// TIA Portal V17 export
// export: Created 2024-08-29T18:23:43.8090158Z, ExportSetting WithDefaults, DisplayName Totally Integrated Automation Portal, DisplayVersion V17 Update 7, DisplayName TIA Portal Openness, DisplayVersion V17 Update 7, DisplayName TIA Portal Version Control Interface, DisplayVersion V17, DisplayName SINAMICS Startdrive Advanced, DisplayVersion V17 SP2, DisplayName SINAMICS Startdrive G110M, G120, G120C, G120D, G120P, G115D, DisplayVersion V17 SP2, DisplayName SINAMICS Startdrive G130, G150, S120, S150, SINAMICS MV, S210, DisplayVersion V17 SP2, DisplayName STEP 7 Professional, DisplayVersion V17 Update 7, DisplayName STEP 7 Safety, DisplayVersion V17 Update 6, DisplayName WinCC Advanced / Unified PC, DisplayVersion V17 Update 7
DATA_BLOCK "analog"   // DB3
{ S7_Optimized_Access := 'TRUE' }
VERSION : 0.1
// stored: AutoNumber false, DBAccessibleFromOPCUA true, DBAccessibleFromWebserver true, IsOnlyStoredInLoadMemory false, IsRetainMemResEnabled false, IsWriteProtectedInAS false, MemoryReserve 100
   VAR RETAIN
      value1 : Array[0..32] of Real;   // Setpoint del valor analógico 1 [modelo]
      low1 : Array[0..32] of Real;   // Valor bajo del valor analógico 1 [modelo]
      high1 : Array[0..32] of Real;   // Valor alto del valor analógico 1 [modelo]
      value2 : Array[0..32] of Real;
      low2 : Array[0..32] of Real;
      high2 : Array[0..32] of Real;
      value3 : Array[0..32] of Real;
      low3 : Array[0..32] of Real;
      high3 : Array[0..32] of Real;
      value4 : Array[0..32] of Real;
      low4 : Array[0..32] of Real;
      high4 : Array[0..32] of Real;
      value5 : Array[0..32] of Real;
      low5 : Array[0..32] of Real;
      high5 : Array[0..32] of Real;
      value6 : Array[0..32] of Real;
      low6 : Array[0..32] of Real;
      high6 : Array[0..32] of Real;
      value7 : Array[0..32] of Real;
      low7 : Array[0..32] of Real;
      high7 : Array[0..32] of Real;
      value8 : Array[0..32] of Real;
      low8 : Array[0..32] of Real;
      high8 : Array[0..32] of Real;
      value9 : Array[0..32] of Real;
      low9 : Array[0..32] of Real;
      high9 : Array[0..32] of Real;
      value10 : Array[0..32] of Real;
      low10 : Array[0..32] of Real;
      high10 : Array[0..32] of Real;
      text : Array[0..10] of String;
      analog1 : Bool := TRUE;
      analog2 : Bool := TRUE;
      analog3 : Bool := TRUE;
      analog4 : Bool := TRUE;
      analog5 : Bool := FALSE;
      analog6 : Bool := FALSE;
   END_VAR
   VAR
      visibility : Array[0..6] of Bool;
      current1 : Int := 0;
      current2 : Int := 0;
      current3 : Int := 0;
      current4 : Int := 0;
      current5 : Int := 0;
      current6 : Int := 0;
      laserConstant : Real := 0.005802801;
      okDistance : Bool := FALSE;
      nest1 : Array[0..5] of Int;
      nest2 : Array[0..5] of Int;
      nest3 : Array[0..5] of Int;
      nest4 : Array[0..5] of Int;
      motorCounter : Int := 1600;
   END_VAR
   VAR RETAIN
      motorQuantity : Int := 0;
   END_VAR
   VAR
      analogReading1 : Array[0..9] of Real;
      analogReading2 : Array[0..9] of Real;
      leftLoadCellMaxValueObtained : Real := 0.0;
      rightLoadCellMaxValueObtained : Real := 0.0;
   END_VAR
BEGIN
   value1[0..3] := -63.9458;
   value1[4] := -16.86112;
   value1[5..8] := -63.9458;
   value1[9..14] := 131.4746;
   value1[15] := 340.0;
   value1[16] := -17.19834;
   value1[17..19] := 131.4746;
   value1[20..32] := 0.0;
   low1[0..2] := -1.0;
   low1[3] := 120.0;
   low1[4] := 154.0;
   low1[5] := 100.0;
   low1[6..8] := 72.0;
   low1[9..13] := 120.0;
   low1[14] := 153.0;
   low1[15] := 0.0;
   low1[16..17] := 120.0;
   low1[18] := 154.0;
   low1[19] := 120.0;
   low1[20..32] := 0.0;
   high1[0..2] := 2.0;
   high1[3] := 5.0;
   high1[4] := 2.0;
   high1[5] := 110.0;
   high1[6..8] := 76.0;
   high1[9..13] := 5.0;
   high1[14] := 2.0;
   high1[15] := 41.1;
   high1[16..17] := 5.0;
   high1[18] := 2.0;
   high1[19] := 5.0;
   high1[20..32] := 0.0;
   value2[0..3] := -65.29469;
   value2[4] := -17.51449;
   value2[5..8] := -65.29469;
   value2[9..14] := 131.4746;
   value2[15] := 340.0;
   value2[16] := -17.40911;
   value2[17..19] := 131.4746;
   value2[20..32] := 0.0;
   low2[0..2] := -1.0;
   low2[3] := 60.0;
   low2[4] := 154.0;
   low2[5] := 100.0;
   low2[6..8] := 60.0;
   low2[9..13] := 0.0;
   low2[14] := 153.0;
   low2[15..17] := 0.0;
   low2[18] := 154.0;
   low2[19..32] := 0.0;
   high2[0..2] := 2.0;
   high2[3] := 75.0;
   high2[4] := 2.0;
   high2[5] := 110.0;
   high2[6..8] := 64.0;
   high2[9..13] := 5.0;
   high2[14] := 2.0;
   high2[15] := 38.7;
   high2[16..17] := 5.0;
   high2[18] := 2.0;
   high2[19] := 5.0;
   high2[20..32] := 0.0;
   value3[0..3] := 16#0000_02E7;
   value3[4] := 16#0000_01DE;
   value3[5..8] := 16#0000_02E7;
   value3[9..14] := 16#0000_01DE;
   value3[15..16] := 16#0000_DDDE;
   value3[17..19] := 16#0000_01DE;
   value3[20..32] := 0.0;
   low3[0..2] := 200.0;
   low3[3] := 40.0;
   low3[4] := 0.0;
   low3[5] := 200.0;
   low3[6..8] := 40.0;
   low3[9..32] := 0.0;
   high3[0..2] := 500.0;
   high3[3] := 250.0;
   high3[4] := 0.0;
   high3[5] := 210.0;
   high3[6..8] := 250.0;
   high3[9..32] := 0.0;
   value4[0..19] := 40.0;
   value4[20..32] := 0.0;
   low4[0..2] := 200.0;
   low4[3] := 40.0;
   low4[4] := 0.0;
   low4[5] := 200.0;
   low4[6..8] := 40.0;
   low4[9..32] := 0.0;
   high4[0..2] := 500.0;
   high4[3] := 250.0;
   high4[4] := 3.0;
   high4[5] := 210.0;
   high4[6..8] := 250.0;
   high4[9..19] := 3.0;
   high4[20..32] := 0.0;
   value5[0..14] := 3.0;
   value5[15] := 8.0;
   value5[16..19] := 3.0;
   value5[20..32] := 0.0;
   low5[0..32] := 0.0;
   high5[0..19] := 59.0;
   high5[20..32] := 0.0;
   value6[0..32] := 0.0;
   low6[0..32] := 0.0;
   high6[0..32] := 0.0;
   value7[0..3] := -65.29469;
   value7[4] := -16.90327;
   value7[5..8] := -65.29469;
   value7[9..14] := -16.86112;
   value7[15] := 0.0;
   value7[16] := -17.19834;
   value7[17..19] := -16.86112;
   value7[20..32] := 0.0;
   low7[0..3] := 142.0;
   low7[4] := 125.0;
   low7[5..8] := 142.0;
   low7[9..13] := 0.0;
   low7[14] := 26.0;
   low7[15..17] := 0.0;
   low7[18] := 128.0;
   low7[19..32] := 0.0;
   high7[0..3] := 2.0;
   high7[4] := 3.0;
   high7[5..13] := 2.0;
   high7[14] := 5.0;
   high7[15] := 0.0;
   high7[16..19] := 2.0;
   high7[20..32] := 0.0;
   value8[0..3] := -65.29469;
   value8[4] := -17.17727;
   value8[5..8] := -65.29469;
   value8[9..14] := -17.17727;
   value8[15] := 0.0;
   value8[16] := -17.51449;
   value8[17..19] := -17.17727;
   value8[20..32] := 0.0;
   low8[0..3] := 142.0;
   low8[4] := 125.0;
   low8[5..8] := 142.0;
   low8[9..13] := 0.0;
   low8[14] := 26.0;
   low8[15..17] := 0.0;
   low8[18] := 128.0;
   low8[19..32] := 0.0;
   high8[0..3] := 2.0;
   high8[4] := 3.0;
   high8[5..13] := 2.0;
   high8[14] := 5.0;
   high8[15] := 0.0;
   high8[16..19] := 2.0;
   high8[20..32] := 0.0;
   value9[0..3] := 1.348892;
   value9[4] := 0.6533699;
   value9[5..8] := 1.348892;
   value9[9..32] := 0.0;
   low9[0..32] := 0.0;
   high9[0..3] := 0.0;
   high9[4] := 2.0;
   high9[5..13] := 0.0;
   high9[14] := 2.0;
   high9[15..17] := 0.0;
   high9[18] := 2.0;
   high9[19..32] := 0.0;
   value10[0..3] := 0.0;
   value10[4] := 0.2739925;
   value10[5..8] := 0.0;
   value10[9..14] := 0.3161469;
   value10[15..16] := 0.0;
   value10[17..19] := 0.3161469;
   value10[20..32] := 0.0;
   low10[0..32] := 0.0;
   high10[0..17] := 0.0;
   high10[18] := 2.0;
   high10[19..32] := 0.0;
   text[0] := '';
   text[1] := 'Distancia Izquierda';
   text[2] := 'Distancia Derecha';
   text[3] := 'Esfuerzo Izquierdo';
   text[4] := 'Esfuerzo Derecho';
   text[5..6] := '';
   text[7] := 'Final izquierdo';
   text[8] := 'Final derecho';
   text[9] := 'Alineacion inicial';
   text[10] := 'Alineacion final';
   visibility[0] := FALSE;
   visibility[1..4] := TRUE;
   visibility[5..6] := FALSE;
   nest1[0..5] := 0;
   nest2[0..5] := 0;
   nest3[0..5] := 0;
   nest4[0..5] := 0;
   analogReading1[0..2] := 58.96373;
   analogReading1[3] := 0.4987493;
   analogReading1[4] := 0.0;
   analogReading1[5..9] := 58.96373;
   analogReading2[0..9] := 0.0;
END_DATA_BLOCK
